TYPE ST_ErrorStruct :
STRUCT
	b_ErrorActive	:BOOL;
	s_Severity 		:STRING(20);
	w_ID			:WORD;
	s_Message		:STRING(100);
	s_DateError		:STRING(20);
	s_TimeError		:STRING(20);
	s_TimeCleared	:STRING(20);
	b_SMSEnable		:BOOL;
END_STRUCT
END_TYPE

(* stored: Version 1.1.0.1, ProductVersion 3.1.4026.18
   DUT ST_ErrorStruct: Id {490887b5-fdfd-4614-997f-d2dcc0985e9c} *)
